RoboDK station: cylinder_surface_test.rdk

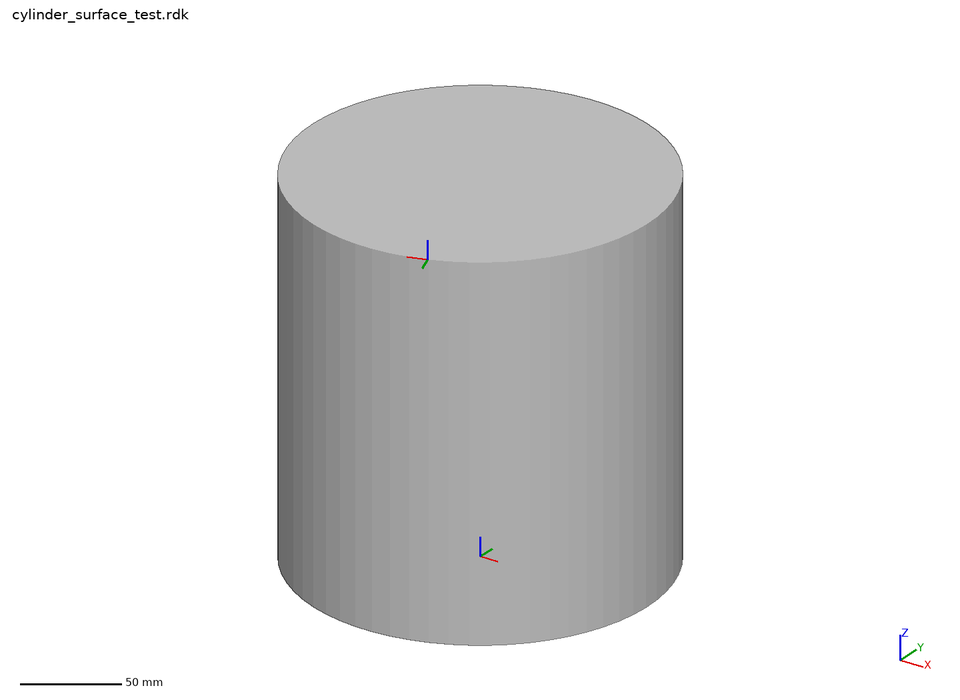
[picture v0: the station drawn from its stored meshes, robots at their saved joint values, targets as dots, program paths as lines]
Station cylinder_surface_test (saved by RoboDK 5.0.0). Poses are relative to the parent item; angles as X-Y-Z fixed-axis rotations.
  - frame Frame 1 at (0, 0, 0) mm
    - object Cylinder100_210 at (0, 0, 0) mm, size 200 x 199.7 x 210 mm, geometry from Cylinder100_210.step
    - frame Frame 2 at (34.2, -93.97, 210) mm, rotated rx 0 ry 0 rz -160 deg
